PROGRAM PRG_LARS_SynchroAggregation
VAR
	rtrigNewOuterArrived					: R_TRIG;
	bNewOuterIsProccesing				: BOOL;
	tonValidationTimout					: TON;
	bValidationTimeout					: BOOL;
	bValidationTimeoutReset				: BOOL;
	fbTimeoutCounter						: CTU;
	nCount									: WORD;

	fbInterimCamera						: FB_SCANNER_CameraSelect;
	(*stInterimCameraOptions				: ST_SCANNER_Options := (eScannerType := E_MV_440SR_FULL, nImageBuffer := 1, nExpectedResp := 2);*)
	fbInterimCameraEvaluation			: FB_SCANNER_Evaluation;

	nInterimCameraID						: UINT;
	bInterimCameraTrigger				: BOOL;
	fbInterimCameraOut					: FB_OUTER_InterimCameraOut;

	fbOuterValidationCamera				: FB_SCANNER_CameraSelect;
	(*stOuterValidationCameraOptions		: ST_SCANNER_Options := (eScannerType := E_MV_420_FULL, nImageBuffer := 1, nExpectedResp := 2);*)
	fbOuterValidationEvaluation			: FB_SCANNER_Evaluation;

	fbCheckForDuplicateOuterValidation	: FB_OUTER_CheckDuplicateStatus;

	rtrigOuterValidationCameraDone	: R_TRIG;
	rtrigInterimCameraDone			: R_TRIG;
	bOuterValidationCameraDone		: BOOL;
	bInterimCameraDone				: BOOL;
	bDataReadyForValidation			: BOOL;
	bQAReject							: BOOL;

	aLastImageDataString				: ARRAY[1..2] OF T_PACK_Barcode;
	sLastImageLableString				: T_OUTER_Barcode;

	fbPerformance							: FB_Interval;
	fbMoveOuterData						: FB_OUTER_MoveOuterStatus;
	fbCompleteOuterFromOCV			: FB_OUTER_CompleteDataFromDB_DoubleCam;
	fbMETSValidateOuterForReject			: FB_OUTER_ValidateOuterForReject;
	tofValidateOuterDoneForHMI			: TOF;
	fbMasterListUpdate					: FB_OUTER_MasterListUpdate;

	stLastOuterCompleted				: ST_OUTER_Status;
	sLastReadOuterBarcode			: T_OUTER_Barcode;
	sLastReadConfPackCode1			: T_PACK_Barcode;
	sLastReadConfPackCode2 			: T_PACK_Barcode;
	nOutersCompleted					: UDINT;
	bDoneInfo							: BOOL;

	rtrigSetOuterValidationOK			: R_TRIG;
	rtrigSetOuterValidationNOK		: R_TRIG;

	rsOuterRejectStation 				: RS;
	rsOuterRejectConfirmation 		: RS;

	rtrigResetValidationStatus			: R_TRIG;

	sRejectCode						: STRING(255);
	fbArchiveInvalidOuters			: FB_OUTER_ArchiveInvalidOuters;
	aReasonForReject					: ARRAY[0..50] OF STRING(255);
	bClearList							: BOOL;

	fbOuterProduced					: FB_KPI_GenericEfficiency;
	fbOuterInspection					: FB_KPI_OutersEfficiency;

	fbOuterLevelCounter				: FB_KPI_OuterLevelCounter;

	fbQARejectCounter				: FB_CTU32;
	fbOuterValidationIndexOK			: FB_CTU32;

	ctuConsecutiveOuterRejects		: CTU;
	nActualCount						: WORD;
END_VAR
VAR // added by the converter: edge detectors and wires of the graphical bodies
    _w1 : BOOL;
END_VAR

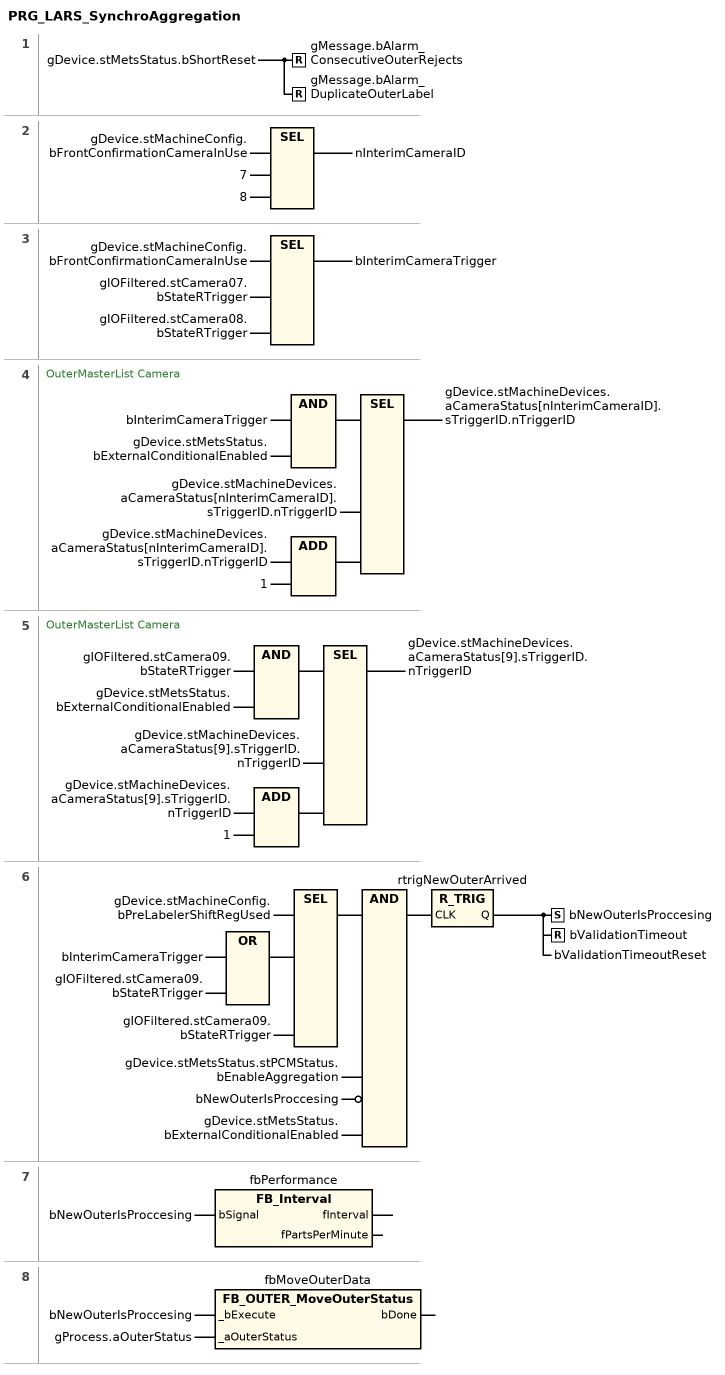
// NETWORK 1
gMessage.bAlarm_ConsecutiveOuterRejects R= gDevice.stMetsStatus.bShortReset;
gMessage.bAlarm_DuplicateOuterLabel R= gDevice.stMetsStatus.bShortReset;

// NETWORK 2
nInterimCameraID := SEL(gDevice.stMachineConfig.bFrontConfirmationCameraInUse, 7, 8);

// NETWORK 3
bInterimCameraTrigger := SEL(gDevice.stMachineConfig.bFrontConfirmationCameraInUse, gIOFiltered.stCamera07.bStateRTrigger, gIOFiltered.stCamera08.bStateRTrigger);

// NETWORK 4
// OuterMasterList Camera
gDevice.stMachineDevices.aCameraStatus[nInterimCameraID].sTriggerID.nTriggerID := SEL(bInterimCameraTrigger AND gDevice.stMetsStatus.bExternalConditionalEnabled, gDevice.stMachineDevices.aCameraStatus[nInterimCameraID].sTriggerID.nTriggerID, gDevice.stMachineDevices.aCameraStatus[nInterimCameraID].sTriggerID.nTriggerID + 1);

// NETWORK 5
// OuterMasterList Camera
gDevice.stMachineDevices.aCameraStatus[9].sTriggerID.nTriggerID := SEL(gIOFiltered.stCamera09.bStateRTrigger AND gDevice.stMetsStatus.bExternalConditionalEnabled, gDevice.stMachineDevices.aCameraStatus[9].sTriggerID.nTriggerID, gDevice.stMachineDevices.aCameraStatus[9].sTriggerID.nTriggerID + 1);

// NETWORK 6
rtrigNewOuterArrived(CLK := SEL(gDevice.stMachineConfig.bPreLabelerShiftRegUsed, bInterimCameraTrigger OR gIOFiltered.stCamera09.bStateRTrigger, gIOFiltered.stCamera09.bStateRTrigger) AND gDevice.stMetsStatus.stPCMStatus.bEnableAggregation AND NOT bNewOuterIsProccesing AND gDevice.stMetsStatus.bExternalConditionalEnabled); // R_TRIG
bNewOuterIsProccesing S= rtrigNewOuterArrived.Q;
bValidationTimeout R= rtrigNewOuterArrived.Q;
bValidationTimeoutReset := rtrigNewOuterArrived.Q;

// NETWORK 7
fbPerformance(bSignal := bNewOuterIsProccesing); // FB_Interval

// NETWORK 8
fbMoveOuterData(_bExecute := bNewOuterIsProccesing, _aOuterStatus := gProcess.aOuterStatus); // FB_OUTER_MoveOuterStatus

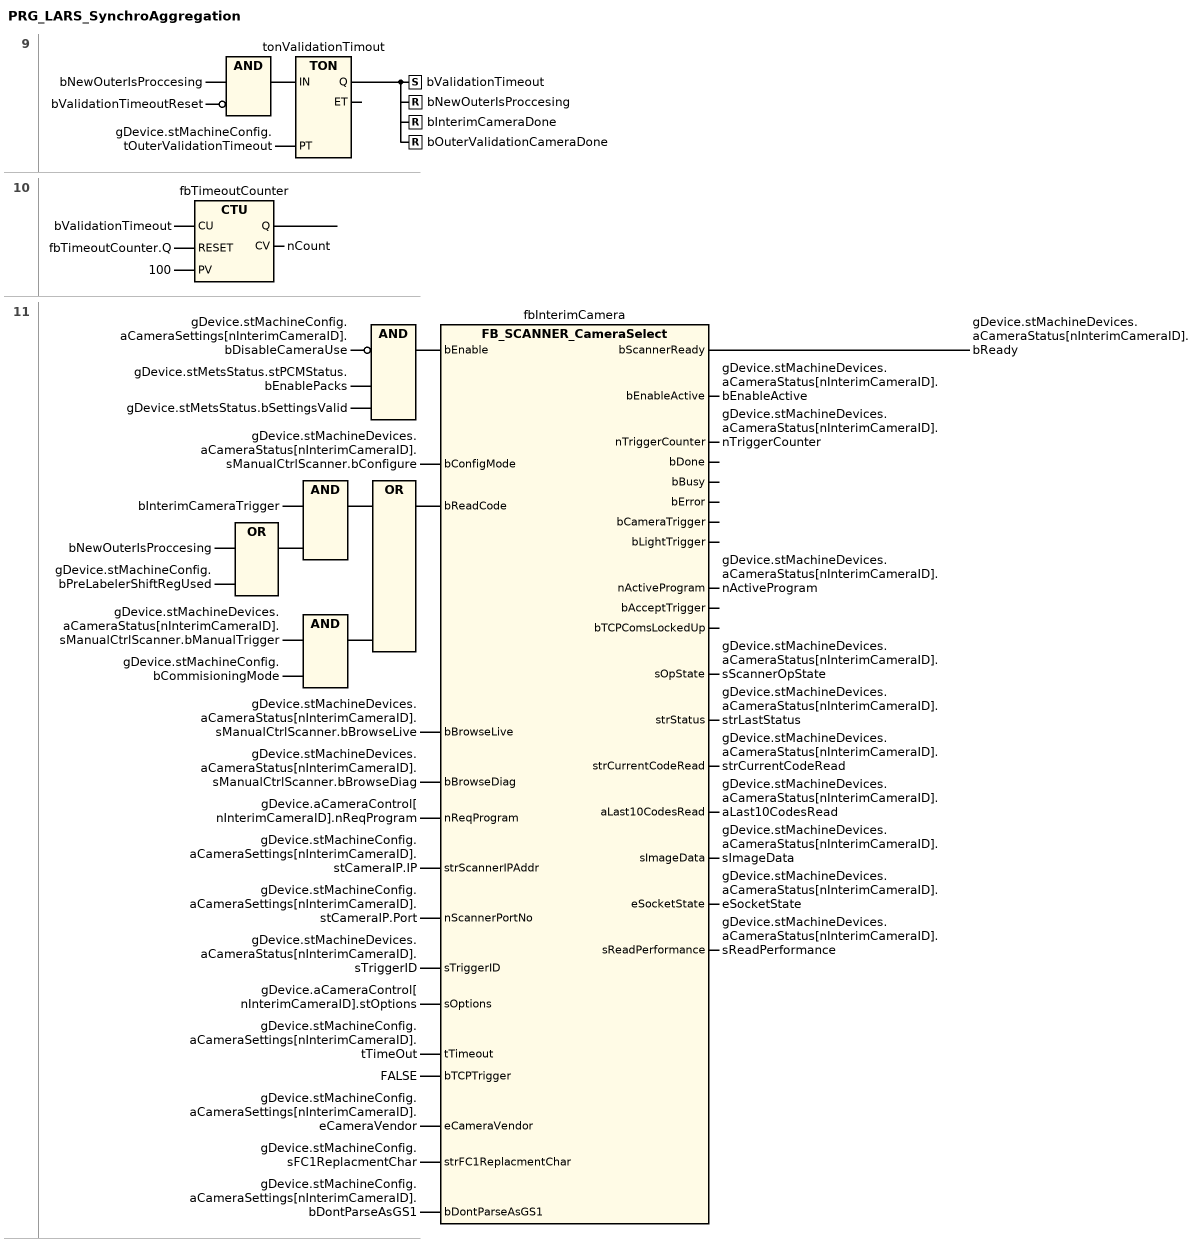
// NETWORK 9
tonValidationTimout(IN := bNewOuterIsProccesing AND NOT bValidationTimeoutReset, PT := gDevice.stMachineConfig.tOuterValidationTimeout); // TON
bValidationTimeout S= tonValidationTimout.Q;
bNewOuterIsProccesing R= tonValidationTimout.Q;
bInterimCameraDone R= tonValidationTimout.Q;
bOuterValidationCameraDone R= tonValidationTimout.Q;

// NETWORK 10
fbTimeoutCounter(CU := bValidationTimeout, RESET := fbTimeoutCounter.Q, PV := 100, CV => nCount); // CTU

// NETWORK 11
fbInterimCamera(
    bEnable := NOT gDevice.stMachineConfig.aCameraSettings[nInterimCameraID].bDisableCameraUse AND gDevice.stMetsStatus.stPCMStatus.bEnablePacks AND gDevice.stMetsStatus.bSettingsValid,
    bConfigMode := gDevice.stMachineDevices.aCameraStatus[nInterimCameraID].sManualCtrlScanner.bConfigure,
    bReadCode := bInterimCameraTrigger AND (bNewOuterIsProccesing OR gDevice.stMachineConfig.bPreLabelerShiftRegUsed) OR gDevice.stMachineDevices.aCameraStatus[nInterimCameraID].sManualCtrlScanner.bManualTrigger AND gDevice.stMachineConfig.bCommisioningMode,
    bBrowseLive := gDevice.stMachineDevices.aCameraStatus[nInterimCameraID].sManualCtrlScanner.bBrowseLive,
    bBrowseDiag := gDevice.stMachineDevices.aCameraStatus[nInterimCameraID].sManualCtrlScanner.bBrowseDiag,
    nReqProgram := gDevice.aCameraControl[nInterimCameraID].nReqProgram,
    strScannerIPAddr := gDevice.stMachineConfig.aCameraSettings[nInterimCameraID].stCameraIP.IP,
    nScannerPortNo := gDevice.stMachineConfig.aCameraSettings[nInterimCameraID].stCameraIP.Port,
    sTriggerID := gDevice.stMachineDevices.aCameraStatus[nInterimCameraID].sTriggerID,
    sOptions := gDevice.aCameraControl[nInterimCameraID].stOptions,
    tTimeout := gDevice.stMachineConfig.aCameraSettings[nInterimCameraID].tTimeOut,
    bTCPTrigger := FALSE,
    eCameraVendor := gDevice.stMachineConfig.aCameraSettings[nInterimCameraID].eCameraVendor,
    strFC1ReplacmentChar := gDevice.stMachineConfig.sFC1ReplacmentChar,
    bDontParseAsGS1 := gDevice.stMachineConfig.aCameraSettings[nInterimCameraID].bDontParseAsGS1,
    bEnableActive => gDevice.stMachineDevices.aCameraStatus[nInterimCameraID].bEnableActive,
    nTriggerCounter => gDevice.stMachineDevices.aCameraStatus[nInterimCameraID].nTriggerCounter,
    nActiveProgram => gDevice.stMachineDevices.aCameraStatus[nInterimCameraID].nActiveProgram,
    sOpState => gDevice.stMachineDevices.aCameraStatus[nInterimCameraID].sScannerOpState,
    strStatus => gDevice.stMachineDevices.aCameraStatus[nInterimCameraID].strLastStatus,
    strCurrentCodeRead => gDevice.stMachineDevices.aCameraStatus[nInterimCameraID].strCurrentCodeRead,
    aLast10CodesRead => gDevice.stMachineDevices.aCameraStatus[nInterimCameraID].aLast10CodesRead,
    sImageData => gDevice.stMachineDevices.aCameraStatus[nInterimCameraID].sImageData,
    eSocketState => gDevice.stMachineDevices.aCameraStatus[nInterimCameraID].eSocketState,
    sReadPerformance => gDevice.stMachineDevices.aCameraStatus[nInterimCameraID].sReadPerformance); // FB_SCANNER_CameraSelect
gDevice.stMachineDevices.aCameraStatus[nInterimCameraID].bReady := fbInterimCamera.bScannerReady;

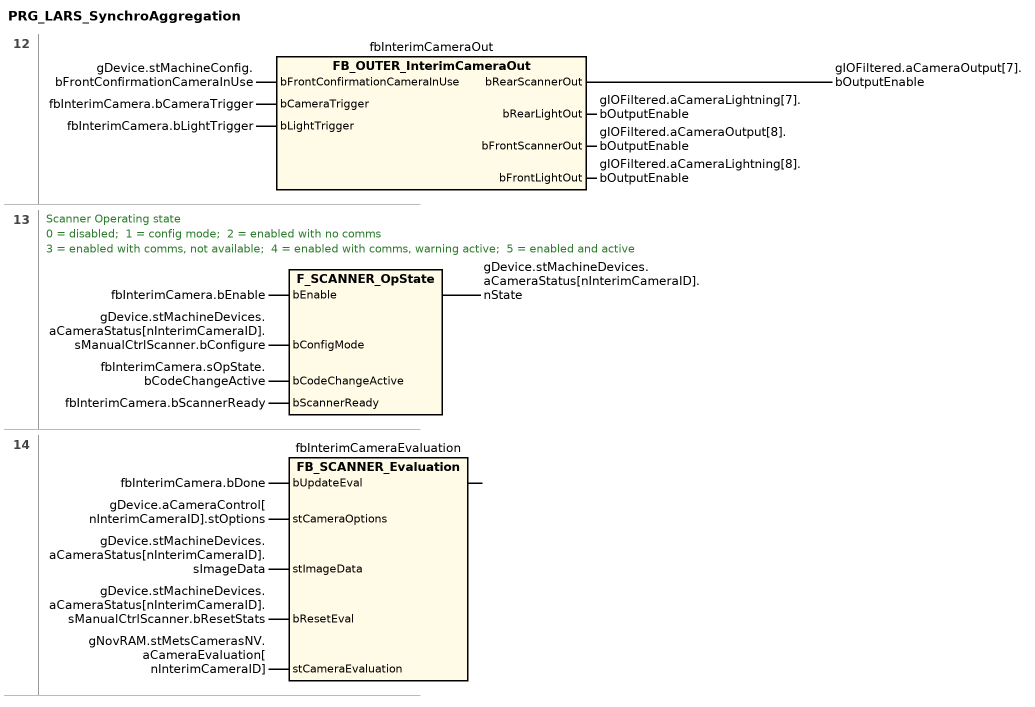
// NETWORK 12
fbInterimCameraOut(
    bFrontConfirmationCameraInUse := gDevice.stMachineConfig.bFrontConfirmationCameraInUse,
    bCameraTrigger := fbInterimCamera.bCameraTrigger,
    bLightTrigger := fbInterimCamera.bLightTrigger,
    bRearLightOut => gIOFiltered.aCameraLightning[7].bOutputEnable,
    bFrontScannerOut => gIOFiltered.aCameraOutput[8].bOutputEnable,
    bFrontLightOut => gIOFiltered.aCameraLightning[8].bOutputEnable); // FB_OUTER_InterimCameraOut
gIOFiltered.aCameraOutput[7].bOutputEnable := fbInterimCameraOut.bRearScannerOut;

// NETWORK 13
// 					Scanner Operating state
// 0 = disabled;  1 = config mode;  2 = enabled with no comms
// 3 = enabled with comms, not available;  4 = enabled with comms, warning active;  5 = enabled and active
//
gDevice.stMachineDevices.aCameraStatus[nInterimCameraID].nState := F_SCANNER_OpState(bEnable := fbInterimCamera.bEnable, bConfigMode := gDevice.stMachineDevices.aCameraStatus[nInterimCameraID].sManualCtrlScanner.bConfigure, bCodeChangeActive := fbInterimCamera.sOpState.bCodeChangeActive, bScannerReady := fbInterimCamera.bScannerReady);

// NETWORK 14
fbInterimCameraEvaluation(
    bUpdateEval := fbInterimCamera.bDone,
    stCameraOptions := gDevice.aCameraControl[nInterimCameraID].stOptions,
    stImageData := gDevice.stMachineDevices.aCameraStatus[nInterimCameraID].sImageData,
    bResetEval := gDevice.stMachineDevices.aCameraStatus[nInterimCameraID].sManualCtrlScanner.bResetStats,
    stCameraEvaluation := gNovRAM.stMetsCamerasNV.aCameraEvaluation[nInterimCameraID]); // FB_SCANNER_Evaluation

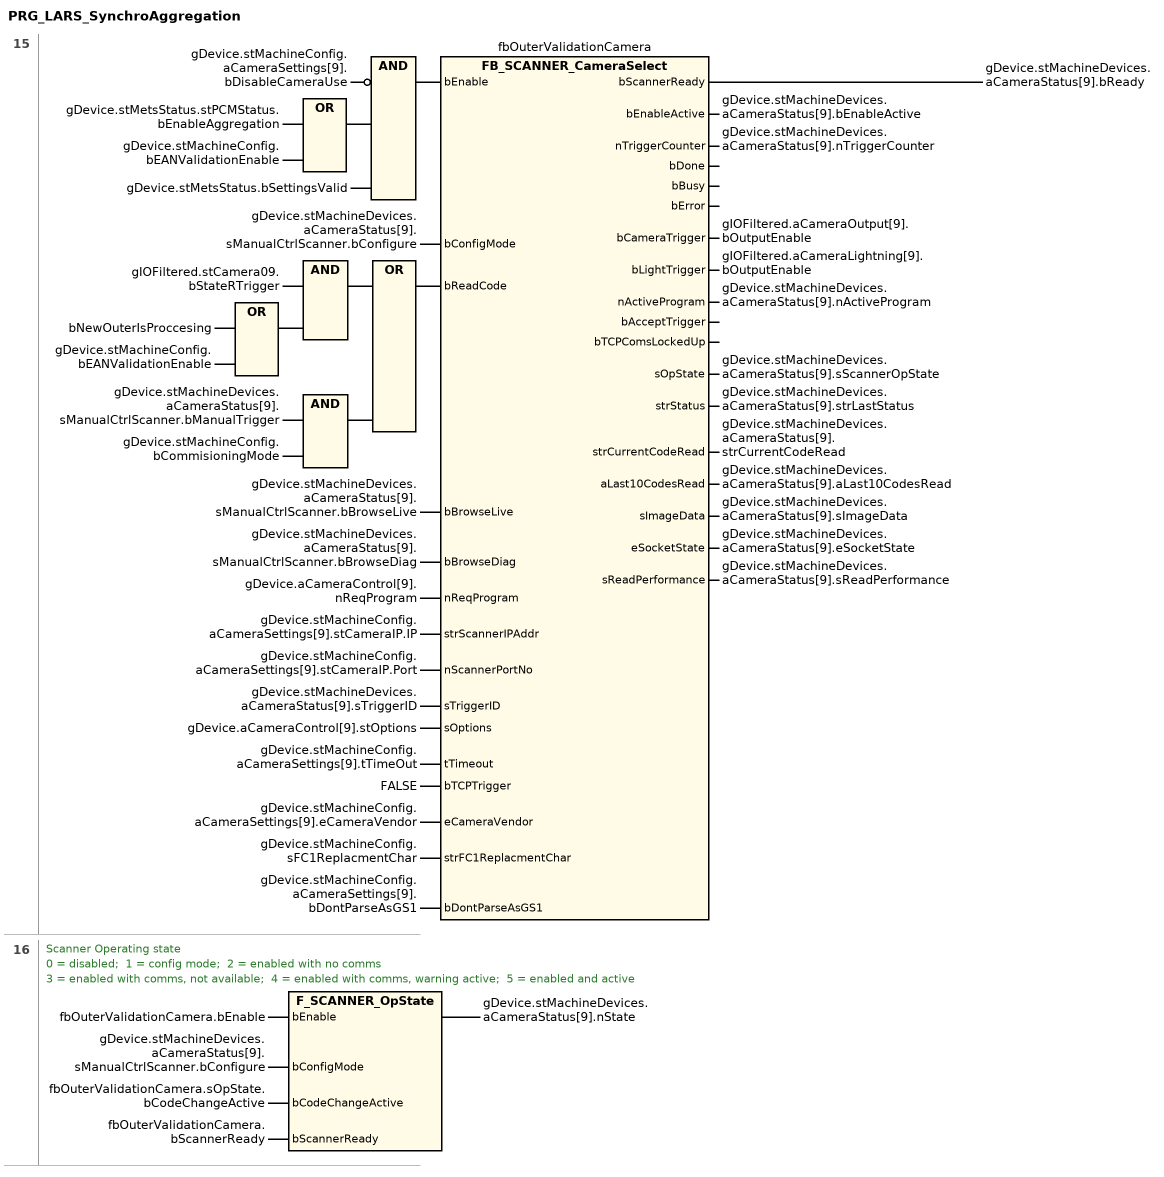
// NETWORK 15
fbOuterValidationCamera(
    bEnable := NOT gDevice.stMachineConfig.aCameraSettings[9].bDisableCameraUse AND (gDevice.stMetsStatus.stPCMStatus.bEnableAggregation OR gDevice.stMachineConfig.bEANValidationEnable) AND gDevice.stMetsStatus.bSettingsValid,
    bConfigMode := gDevice.stMachineDevices.aCameraStatus[9].sManualCtrlScanner.bConfigure,
    bReadCode := gIOFiltered.stCamera09.bStateRTrigger AND (bNewOuterIsProccesing OR gDevice.stMachineConfig.bEANValidationEnable) OR gDevice.stMachineDevices.aCameraStatus[9].sManualCtrlScanner.bManualTrigger AND gDevice.stMachineConfig.bCommisioningMode,
    bBrowseLive := gDevice.stMachineDevices.aCameraStatus[9].sManualCtrlScanner.bBrowseLive,
    bBrowseDiag := gDevice.stMachineDevices.aCameraStatus[9].sManualCtrlScanner.bBrowseDiag,
    nReqProgram := gDevice.aCameraControl[9].nReqProgram,
    strScannerIPAddr := gDevice.stMachineConfig.aCameraSettings[9].stCameraIP.IP,
    nScannerPortNo := gDevice.stMachineConfig.aCameraSettings[9].stCameraIP.Port,
    sTriggerID := gDevice.stMachineDevices.aCameraStatus[9].sTriggerID,
    sOptions := gDevice.aCameraControl[9].stOptions,
    tTimeout := gDevice.stMachineConfig.aCameraSettings[9].tTimeOut,
    bTCPTrigger := FALSE,
    eCameraVendor := gDevice.stMachineConfig.aCameraSettings[9].eCameraVendor,
    strFC1ReplacmentChar := gDevice.stMachineConfig.sFC1ReplacmentChar,
    bDontParseAsGS1 := gDevice.stMachineConfig.aCameraSettings[9].bDontParseAsGS1,
    bEnableActive => gDevice.stMachineDevices.aCameraStatus[9].bEnableActive,
    nTriggerCounter => gDevice.stMachineDevices.aCameraStatus[9].nTriggerCounter,
    bCameraTrigger => gIOFiltered.aCameraOutput[9].bOutputEnable,
    bLightTrigger => gIOFiltered.aCameraLightning[9].bOutputEnable,
    nActiveProgram => gDevice.stMachineDevices.aCameraStatus[9].nActiveProgram,
    sOpState => gDevice.stMachineDevices.aCameraStatus[9].sScannerOpState,
    strStatus => gDevice.stMachineDevices.aCameraStatus[9].strLastStatus,
    strCurrentCodeRead => gDevice.stMachineDevices.aCameraStatus[9].strCurrentCodeRead,
    aLast10CodesRead => gDevice.stMachineDevices.aCameraStatus[9].aLast10CodesRead,
    sImageData => gDevice.stMachineDevices.aCameraStatus[9].sImageData,
    eSocketState => gDevice.stMachineDevices.aCameraStatus[9].eSocketState,
    sReadPerformance => gDevice.stMachineDevices.aCameraStatus[9].sReadPerformance); // FB_SCANNER_CameraSelect
gDevice.stMachineDevices.aCameraStatus[9].bReady := fbOuterValidationCamera.bScannerReady;

// NETWORK 16
// 					Scanner Operating state
// 0 = disabled;  1 = config mode;  2 = enabled with no comms
// 3 = enabled with comms, not available;  4 = enabled with comms, warning active;  5 = enabled and active
//
gDevice.stMachineDevices.aCameraStatus[9].nState := F_SCANNER_OpState(bEnable := fbOuterValidationCamera.bEnable, bConfigMode := gDevice.stMachineDevices.aCameraStatus[9].sManualCtrlScanner.bConfigure, bCodeChangeActive := fbOuterValidationCamera.sOpState.bCodeChangeActive, bScannerReady := fbOuterValidationCamera.bScannerReady);

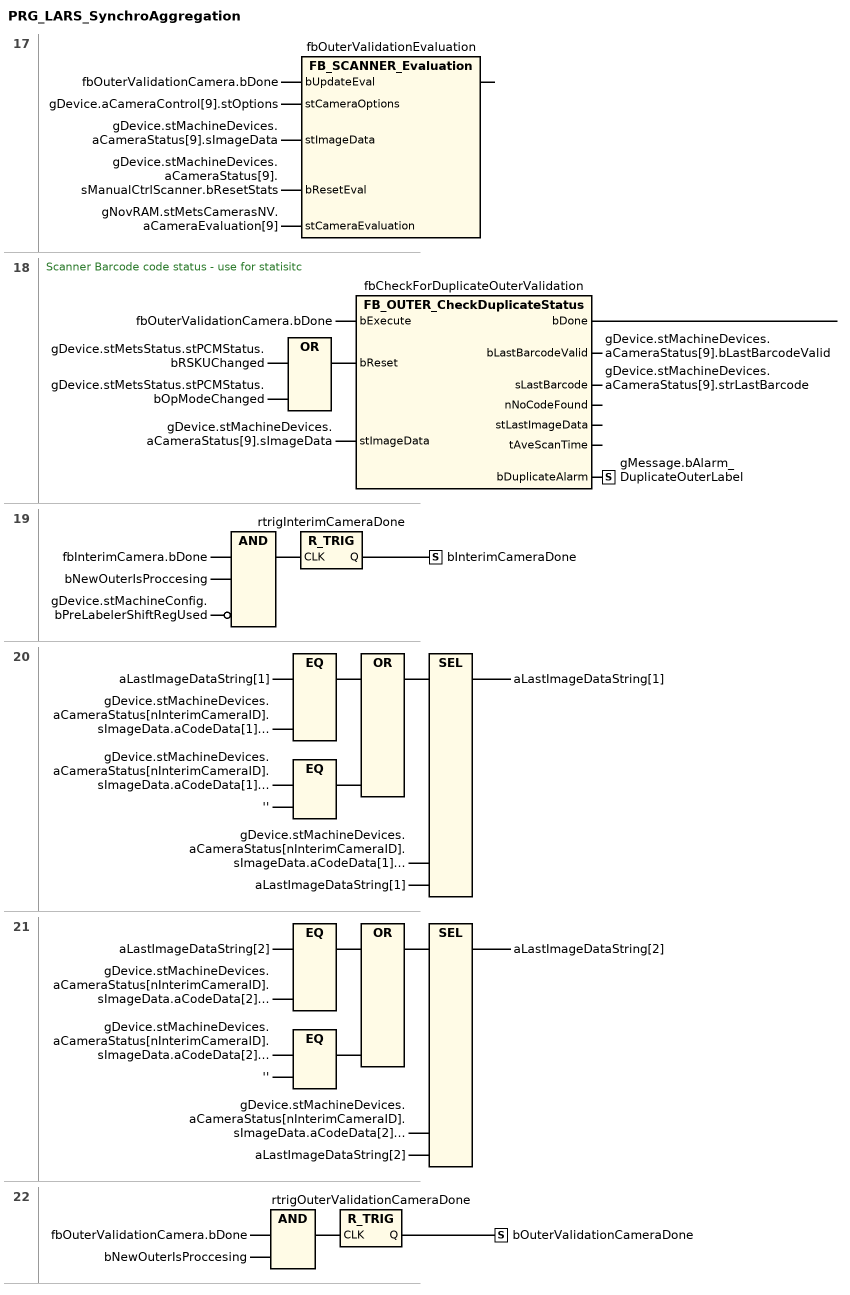
// NETWORK 17
fbOuterValidationEvaluation(
    bUpdateEval := fbOuterValidationCamera.bDone,
    stCameraOptions := gDevice.aCameraControl[9].stOptions,
    stImageData := gDevice.stMachineDevices.aCameraStatus[9].sImageData,
    bResetEval := gDevice.stMachineDevices.aCameraStatus[9].sManualCtrlScanner.bResetStats,
    stCameraEvaluation := gNovRAM.stMetsCamerasNV.aCameraEvaluation[9]); // FB_SCANNER_Evaluation

// NETWORK 18
// Scanner Barcode code status - use for statisitc
fbCheckForDuplicateOuterValidation(
    bExecute := fbOuterValidationCamera.bDone,
    bReset := gDevice.stMetsStatus.stPCMStatus.bRSKUChanged OR gDevice.stMetsStatus.stPCMStatus.bOpModeChanged,
    stImageData := gDevice.stMachineDevices.aCameraStatus[9].sImageData,
    bLastBarcodeValid => gDevice.stMachineDevices.aCameraStatus[9].bLastBarcodeValid,
    sLastBarcode => gDevice.stMachineDevices.aCameraStatus[9].strLastBarcode); // FB_OUTER_CheckDuplicateStatus
gMessage.bAlarm_DuplicateOuterLabel S= fbCheckForDuplicateOuterValidation.bDuplicateAlarm;

// NETWORK 19
rtrigInterimCameraDone(CLK := fbInterimCamera.bDone AND bNewOuterIsProccesing AND NOT gDevice.stMachineConfig.bPreLabelerShiftRegUsed); // R_TRIG
bInterimCameraDone S= rtrigInterimCameraDone.Q;

// NETWORK 20
aLastImageDataString[1] := SEL(aLastImageDataString[1] = gDevice.stMachineDevices.aCameraStatus[nInterimCameraID].sImageData.aCodeData[1].strDataString OR gDevice.stMachineDevices.aCameraStatus[nInterimCameraID].sImageData.aCodeData[1].strDataString = '', gDevice.stMachineDevices.aCameraStatus[nInterimCameraID].sImageData.aCodeData[1].strDataString, aLastImageDataString[1]);

// NETWORK 21
aLastImageDataString[2] := SEL(aLastImageDataString[2] = gDevice.stMachineDevices.aCameraStatus[nInterimCameraID].sImageData.aCodeData[2].strDataString OR gDevice.stMachineDevices.aCameraStatus[nInterimCameraID].sImageData.aCodeData[2].strDataString = '', gDevice.stMachineDevices.aCameraStatus[nInterimCameraID].sImageData.aCodeData[2].strDataString, aLastImageDataString[2]);

// NETWORK 22
rtrigOuterValidationCameraDone(CLK := fbOuterValidationCamera.bDone AND bNewOuterIsProccesing); // R_TRIG
bOuterValidationCameraDone S= rtrigOuterValidationCameraDone.Q;

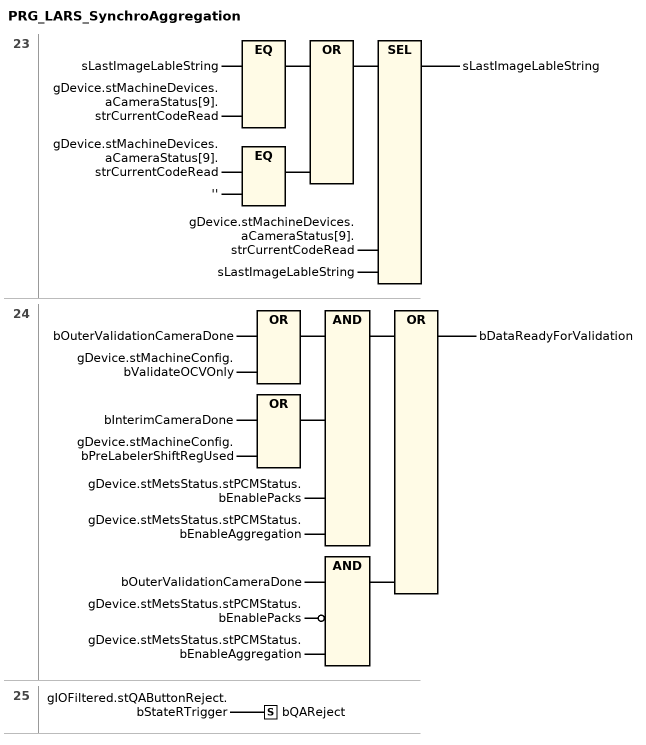
// NETWORK 23
sLastImageLableString := SEL(sLastImageLableString = gDevice.stMachineDevices.aCameraStatus[9].strCurrentCodeRead OR gDevice.stMachineDevices.aCameraStatus[9].strCurrentCodeRead = '', gDevice.stMachineDevices.aCameraStatus[9].strCurrentCodeRead, sLastImageLableString);

// NETWORK 24
bDataReadyForValidation := (bOuterValidationCameraDone OR gDevice.stMachineConfig.bValidateOCVOnly) AND (bInterimCameraDone OR gDevice.stMachineConfig.bPreLabelerShiftRegUsed) AND gDevice.stMetsStatus.stPCMStatus.bEnablePacks AND gDevice.stMetsStatus.stPCMStatus.bEnableAggregation OR bOuterValidationCameraDone AND NOT gDevice.stMetsStatus.stPCMStatus.bEnablePacks AND gDevice.stMetsStatus.stPCMStatus.bEnableAggregation;

// NETWORK 25
bQAReject S= gIOFiltered.stQAButtonReject.bStateRTrigger;

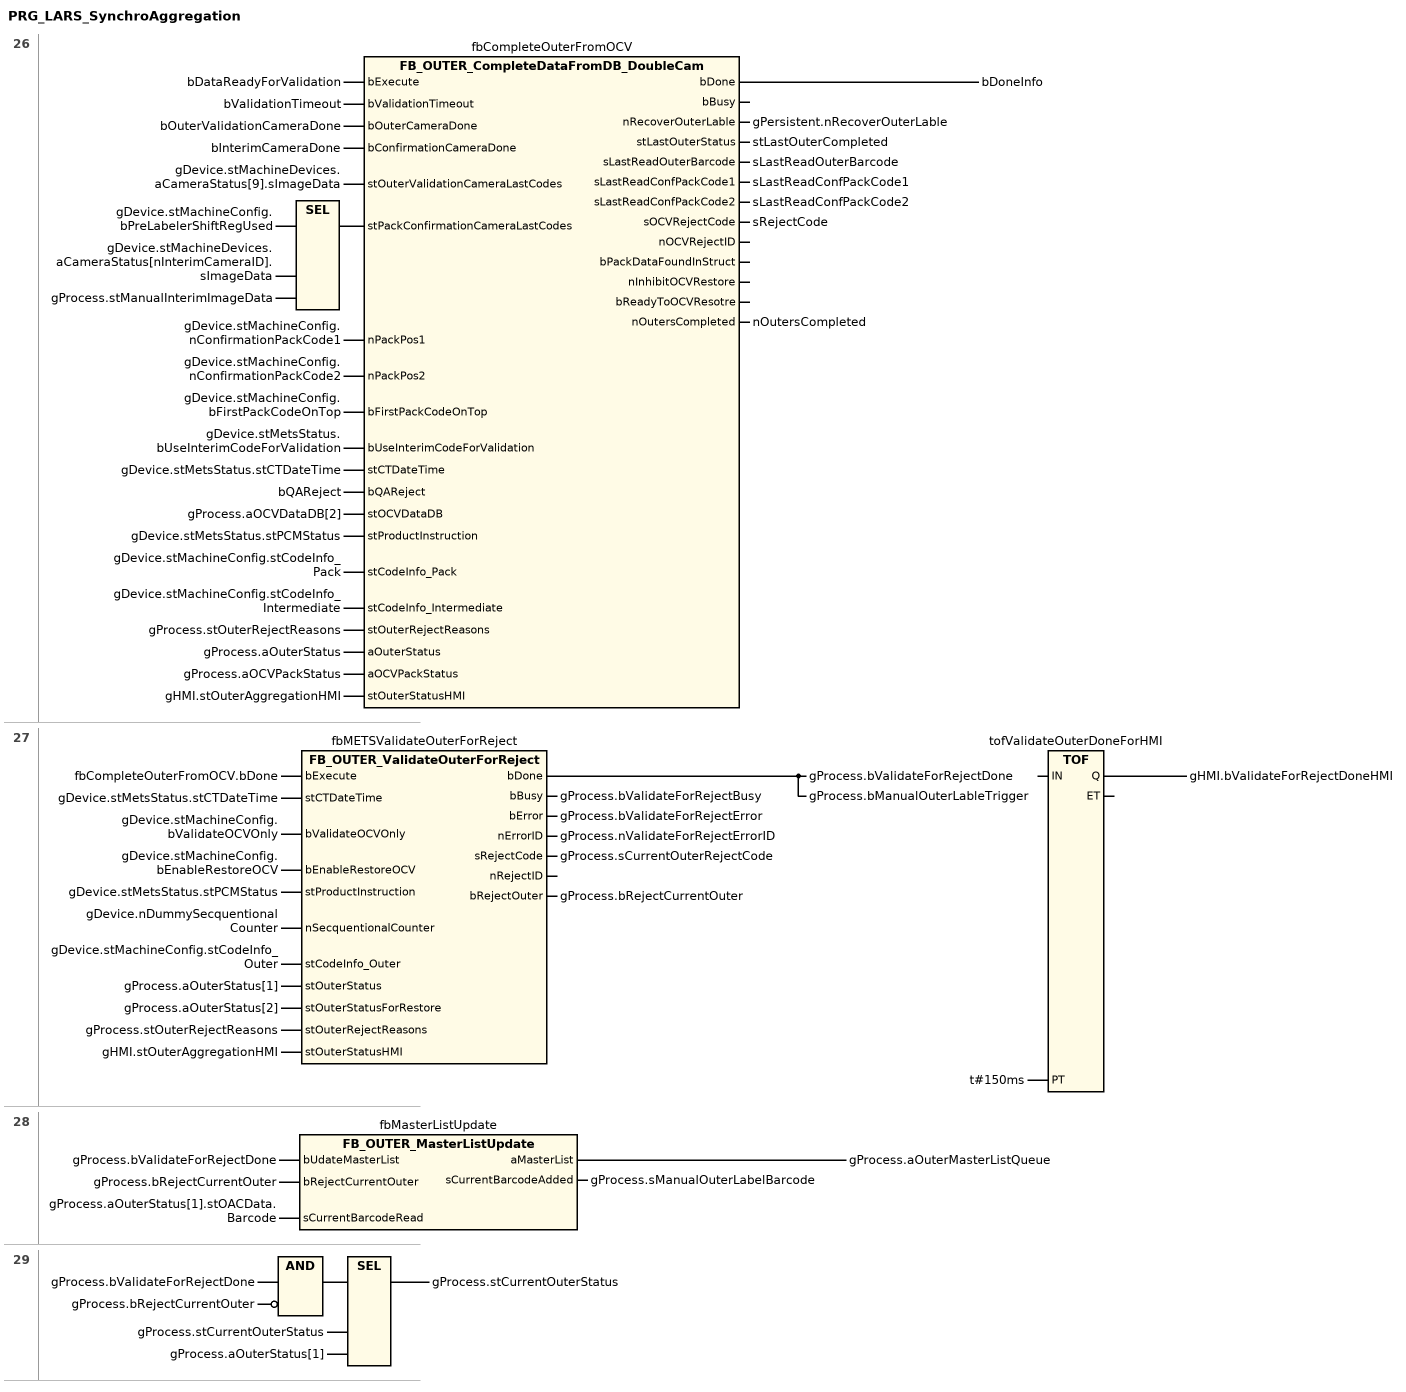
// NETWORK 26
fbCompleteOuterFromOCV(
    bExecute := bDataReadyForValidation,
    bValidationTimeout := bValidationTimeout,
    bOuterCameraDone := bOuterValidationCameraDone,
    bConfirmationCameraDone := bInterimCameraDone,
    stOuterValidationCameraLastCodes := gDevice.stMachineDevices.aCameraStatus[9].sImageData,
    stPackConfirmationCameraLastCodes := SEL(gDevice.stMachineConfig.bPreLabelerShiftRegUsed, gDevice.stMachineDevices.aCameraStatus[nInterimCameraID].sImageData, gProcess.stManualInterimImageData),
    nPackPos1 := gDevice.stMachineConfig.nConfirmationPackCode1,
    nPackPos2 := gDevice.stMachineConfig.nConfirmationPackCode2,
    bFirstPackCodeOnTop := gDevice.stMachineConfig.bFirstPackCodeOnTop,
    bUseInterimCodeForValidation := gDevice.stMetsStatus.bUseInterimCodeForValidation,
    stCTDateTime := gDevice.stMetsStatus.stCTDateTime,
    bQAReject := bQAReject,
    stOCVDataDB := gProcess.aOCVDataDB[2],
    stProductInstruction := gDevice.stMetsStatus.stPCMStatus,
    stCodeInfo_Pack := gDevice.stMachineConfig.stCodeInfo_Pack,
    stCodeInfo_Intermediate := gDevice.stMachineConfig.stCodeInfo_Intermediate,
    stOuterRejectReasons := gProcess.stOuterRejectReasons,
    aOuterStatus := gProcess.aOuterStatus,
    aOCVPackStatus := gProcess.aOCVPackStatus,
    stOuterStatusHMI := gHMI.stOuterAggregationHMI,
    nRecoverOuterLable => gPersistent.nRecoverOuterLable,
    stLastOuterStatus => stLastOuterCompleted,
    sLastReadOuterBarcode => sLastReadOuterBarcode,
    sLastReadConfPackCode1 => sLastReadConfPackCode1,
    sLastReadConfPackCode2 => sLastReadConfPackCode2,
    sOCVRejectCode => sRejectCode,
    nOutersCompleted => nOutersCompleted); // FB_OUTER_CompleteDataFromDB_DoubleCam
bDoneInfo := fbCompleteOuterFromOCV.bDone;

// NETWORK 27
fbMETSValidateOuterForReject(
    bExecute := fbCompleteOuterFromOCV.bDone,
    stCTDateTime := gDevice.stMetsStatus.stCTDateTime,
    bValidateOCVOnly := gDevice.stMachineConfig.bValidateOCVOnly,
    bEnableRestoreOCV := gDevice.stMachineConfig.bEnableRestoreOCV,
    stProductInstruction := gDevice.stMetsStatus.stPCMStatus,
    nSecquentionalCounter := gDevice.nDummySecquentionalCounter,
    stCodeInfo_Outer := gDevice.stMachineConfig.stCodeInfo_Outer,
    stOuterStatus := gProcess.aOuterStatus[1],
    stOuterStatusForRestore := gProcess.aOuterStatus[2],
    stOuterRejectReasons := gProcess.stOuterRejectReasons,
    stOuterStatusHMI := gHMI.stOuterAggregationHMI,
    bBusy => gProcess.bValidateForRejectBusy,
    bError => gProcess.bValidateForRejectError,
    nErrorID => gProcess.nValidateForRejectErrorID,
    sRejectCode => gProcess.sCurrentOuterRejectCode,
    bRejectOuter => gProcess.bRejectCurrentOuter); // FB_OUTER_ValidateOuterForReject
gProcess.bValidateForRejectDone := fbMETSValidateOuterForReject.bDone;
gProcess.bManualOuterLableTrigger := fbMETSValidateOuterForReject.bDone;
tofValidateOuterDoneForHMI(IN := fbMETSValidateOuterForReject.bDone, PT := t#150ms); // TOF
gHMI.bValidateForRejectDoneHMI := tofValidateOuterDoneForHMI.Q;

// NETWORK 28
fbMasterListUpdate(
    bUdateMasterList := gProcess.bValidateForRejectDone,
    bRejectCurrentOuter := gProcess.bRejectCurrentOuter,
    sCurrentBarcodeRead := gProcess.aOuterStatus[1].stOACData.Barcode,
    sCurrentBarcodeAdded => gProcess.sManualOuterLabelBarcode); // FB_OUTER_MasterListUpdate
gProcess.aOuterMasterListQueue := fbMasterListUpdate.aMasterList;

// NETWORK 29
gProcess.stCurrentOuterStatus := SEL(gProcess.bValidateForRejectDone AND NOT gProcess.bRejectCurrentOuter, gProcess.stCurrentOuterStatus, gProcess.aOuterStatus[1]);

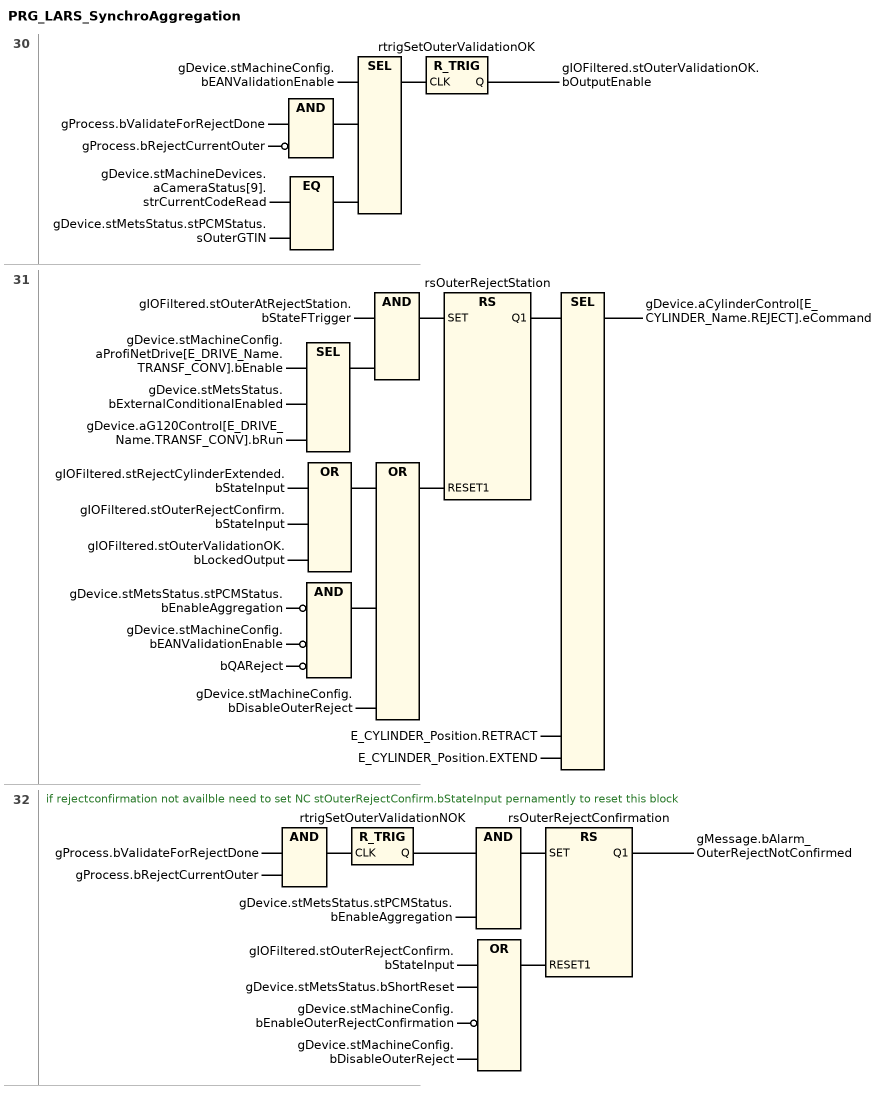
// NETWORK 30
rtrigSetOuterValidationOK(CLK := SEL(gDevice.stMachineConfig.bEANValidationEnable, gProcess.bValidateForRejectDone AND NOT gProcess.bRejectCurrentOuter, gDevice.stMachineDevices.aCameraStatus[9].strCurrentCodeRead = gDevice.stMetsStatus.stPCMStatus.sOuterGTIN)); // R_TRIG
gIOFiltered.stOuterValidationOK.bOutputEnable := rtrigSetOuterValidationOK.Q;

// NETWORK 31
rsOuterRejectStation(SET := gIOFiltered.stOuterAtRejectStation.bStateFTrigger AND SEL(gDevice.stMachineConfig.aProfiNetDrive[E_DRIVE_Name.TRANSF_CONV].bEnable, gDevice.stMetsStatus.bExternalConditionalEnabled, gDevice.aG120Control[E_DRIVE_Name.TRANSF_CONV].bRun), RESET1 := (gIOFiltered.stRejectCylinderExtended.bStateInput OR gIOFiltered.stOuterRejectConfirm.bStateInput OR gIOFiltered.stOuterValidationOK.bLockedOutput) OR NOT gDevice.stMetsStatus.stPCMStatus.bEnableAggregation AND NOT gDevice.stMachineConfig.bEANValidationEnable AND NOT bQAReject OR gDevice.stMachineConfig.bDisableOuterReject); // RS
gDevice.aCylinderControl[E_CYLINDER_Name.REJECT].eCommand := SEL(rsOuterRejectStation.Q1, E_CYLINDER_Position.RETRACT, E_CYLINDER_Position.EXTEND);

// NETWORK 32
// if rejectconfirmation not availble need to set NC stOuterRejectConfirm.bStateInput pernamently to reset this block
rtrigSetOuterValidationNOK(CLK := gProcess.bValidateForRejectDone AND gProcess.bRejectCurrentOuter); // R_TRIG
rsOuterRejectConfirmation(SET := rtrigSetOuterValidationNOK.Q AND gDevice.stMetsStatus.stPCMStatus.bEnableAggregation, RESET1 := gIOFiltered.stOuterRejectConfirm.bStateInput OR gDevice.stMetsStatus.bShortReset OR NOT gDevice.stMachineConfig.bEnableOuterRejectConfirmation OR gDevice.stMachineConfig.bDisableOuterReject); // RS
gMessage.bAlarm_OuterRejectNotConfirmed := rsOuterRejectConfirmation.Q1;

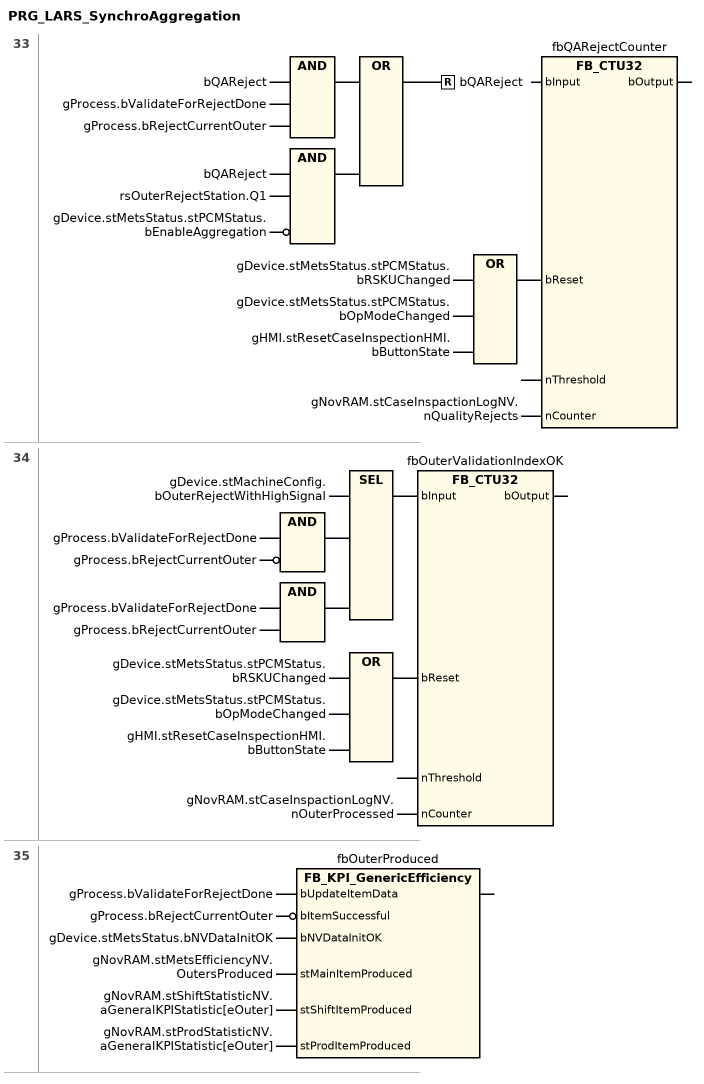
// NETWORK 33
_w1 := bQAReject AND gProcess.bValidateForRejectDone AND gProcess.bRejectCurrentOuter OR bQAReject AND rsOuterRejectStation.Q1 AND NOT gDevice.stMetsStatus.stPCMStatus.bEnableAggregation;
bQAReject R= _w1;
fbQARejectCounter(
    bInput := _w1,
    bReset := gDevice.stMetsStatus.stPCMStatus.bRSKUChanged OR gDevice.stMetsStatus.stPCMStatus.bOpModeChanged OR gHMI.stResetCaseInspectionHMI.bButtonState,
    nCounter := gNovRAM.stCaseInspactionLogNV.nQualityRejects); // FB_CTU32

// NETWORK 34
fbOuterValidationIndexOK(
    bInput := SEL(gDevice.stMachineConfig.bOuterRejectWithHighSignal, gProcess.bValidateForRejectDone AND NOT gProcess.bRejectCurrentOuter, gProcess.bValidateForRejectDone AND gProcess.bRejectCurrentOuter),
    bReset := gDevice.stMetsStatus.stPCMStatus.bRSKUChanged OR gDevice.stMetsStatus.stPCMStatus.bOpModeChanged OR gHMI.stResetCaseInspectionHMI.bButtonState,
    nCounter := gNovRAM.stCaseInspactionLogNV.nOuterProcessed); // FB_CTU32

// NETWORK 35
fbOuterProduced(
    bUpdateItemData := gProcess.bValidateForRejectDone,
    bItemSuccessful := NOT gProcess.bRejectCurrentOuter,
    bNVDataInitOK := gDevice.stMetsStatus.bNVDataInitOK,
    stMainItemProduced := gNovRAM.stMetsEfficiencyNV.OutersProduced,
    stShiftItemProduced := gNovRAM.stShiftStatisticNV.aGeneralKPIStatistic[eOuter],
    stProdItemProduced := gNovRAM.stProdStatisticNV.aGeneralKPIStatistic[eOuter]); // FB_KPI_GenericEfficiency

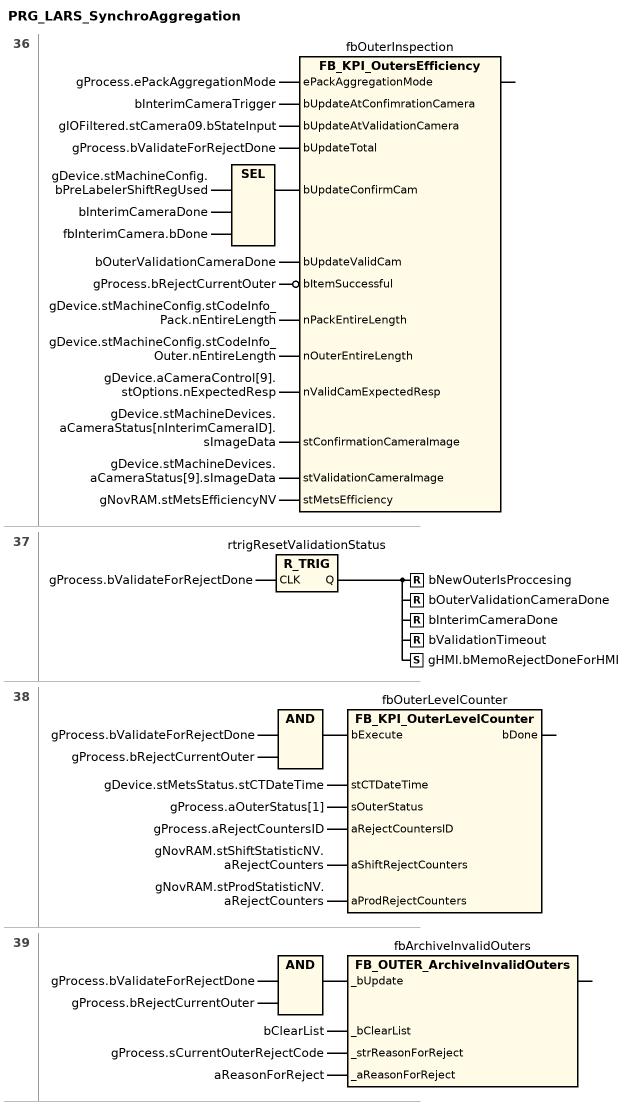
// NETWORK 36
fbOuterInspection(
    ePackAggregationMode := gProcess.ePackAggregationMode,
    bUpdateAtConfimrationCamera := bInterimCameraTrigger,
    bUpdateAtValidationCamera := gIOFiltered.stCamera09.bStateInput,
    bUpdateTotal := gProcess.bValidateForRejectDone,
    bUpdateConfirmCam := SEL(gDevice.stMachineConfig.bPreLabelerShiftRegUsed, bInterimCameraDone, fbInterimCamera.bDone),
    bUpdateValidCam := bOuterValidationCameraDone,
    bItemSuccessful := NOT gProcess.bRejectCurrentOuter,
    nPackEntireLength := gDevice.stMachineConfig.stCodeInfo_Pack.nEntireLength,
    nOuterEntireLength := gDevice.stMachineConfig.stCodeInfo_Outer.nEntireLength,
    nValidCamExpectedResp := gDevice.aCameraControl[9].stOptions.nExpectedResp,
    stConfirmationCameraImage := gDevice.stMachineDevices.aCameraStatus[nInterimCameraID].sImageData,
    stValidationCameraImage := gDevice.stMachineDevices.aCameraStatus[9].sImageData,
    stMetsEfficiency := gNovRAM.stMetsEfficiencyNV); // FB_KPI_OutersEfficiency

// NETWORK 37
rtrigResetValidationStatus(CLK := gProcess.bValidateForRejectDone); // R_TRIG
bNewOuterIsProccesing R= rtrigResetValidationStatus.Q;
bOuterValidationCameraDone R= rtrigResetValidationStatus.Q;
bInterimCameraDone R= rtrigResetValidationStatus.Q;
bValidationTimeout R= rtrigResetValidationStatus.Q;
gHMI.bMemoRejectDoneForHMI S= rtrigResetValidationStatus.Q;

// NETWORK 38
fbOuterLevelCounter(
    bExecute := gProcess.bValidateForRejectDone AND gProcess.bRejectCurrentOuter,
    stCTDateTime := gDevice.stMetsStatus.stCTDateTime,
    sOuterStatus := gProcess.aOuterStatus[1],
    aRejectCountersID := gProcess.aRejectCountersID,
    aShiftRejectCounters := gNovRAM.stShiftStatisticNV.aRejectCounters,
    aProdRejectCounters := gNovRAM.stProdStatisticNV.aRejectCounters); // FB_KPI_OuterLevelCounter

// NETWORK 39
fbArchiveInvalidOuters(
    _bUpdate := gProcess.bValidateForRejectDone AND gProcess.bRejectCurrentOuter,
    _bClearList := bClearList,
    _strReasonForReject := gProcess.sCurrentOuterRejectCode,
    _aReasonForReject := aReasonForReject); // FB_OUTER_ArchiveInvalidOuters

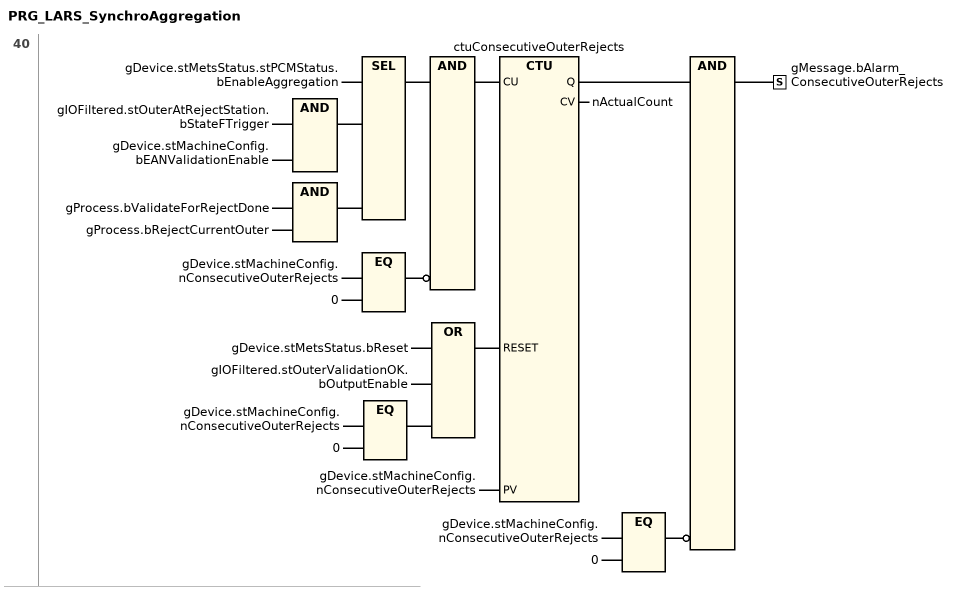
// NETWORK 40
ctuConsecutiveOuterRejects(
    CU := SEL(gDevice.stMetsStatus.stPCMStatus.bEnableAggregation, gIOFiltered.stOuterAtRejectStation.bStateFTrigger AND gDevice.stMachineConfig.bEANValidationEnable, gProcess.bValidateForRejectDone AND gProcess.bRejectCurrentOuter) AND NOT (gDevice.stMachineConfig.nConsecutiveOuterRejects = 0),
    RESET := gDevice.stMetsStatus.bReset OR gIOFiltered.stOuterValidationOK.bOutputEnable OR gDevice.stMachineConfig.nConsecutiveOuterRejects = 0,
    PV := gDevice.stMachineConfig.nConsecutiveOuterRejects,
    CV => nActualCount); // CTU
gMessage.bAlarm_ConsecutiveOuterRejects S= ctuConsecutiveOuterRejects.Q AND NOT (gDevice.stMachineConfig.nConsecutiveOuterRejects = 0);

END_PROGRAM

(* stored: Version 1.1.0.1
   POU PRG_LARS_SynchroAggregation: Id {647cc502-8328-4d9e-9c26-810409adfcbd}, SpecialFunc None *)
